FUNCTION LimitRealNumberToWord : INT
VAR_INPUT
	IN : REAL;
	LowLimit : REAL;
	HighLimit : REAL;
END_VAR
VAR
END_VAR

LimitRealNumberToWord:=REAL_TO_WORD(LimitRealNumber(IN,LowLimit,HighLimit));

END_FUNCTION

(* stored: Version 1.1.0.1, ProductVersion 3.1.4024.15
   POU LimitRealNumberToWord: Id {314fa535-00f5-4ae5-9768-9d048427f829}, SpecialFunc None *)
